TYPE teCTCStep :
(
	FB_CTC_FUNCTIONBLOCK_DISABLED 	:= 0,
	FB_CTC_CONNECTING 				:= 1,
	FB_CTC_DISABLED 				:= 2,
	FB_CTC_ENABLING					:= 21,
	FB_CTC_DISABLING				:= 22,
	FB_CTC_HOME 					:= 3,
	FB_CTC_TEACH 					:= 4,
	FB_CTC_READY 					:= 5,
	FB_CTC_MOVE_OUT 				:= 6,
	FB_CTC_MOVE_IN 					:= 7,
	FB_CTC_MOVE_ABSOLUTE 			:= 8,	
	FB_CTC_MOVE_CONTINUOUS 			:= 9,
	FB_CTC_HALTING 					:= 10,
	FB_CTC_ERROR 					:= 11,
	FB_CTC_RESET 					:= 12
);
END_TYPE

(* stored: Version 1.1.0.1, ProductVersion 3.1.4026.17
   EnumerationTextList teCTCStep: Id {c80fd44a-6701-4cb0-a437-92603f326e26} *)
